INTERFACE I_ControlScheme

END_INTERFACE

(* stored: Version 1.1.0.1, ProductVersion 3.1.4024.6
   Itf I_ControlScheme: Id {f000d3ae-a91a-4047-91a4-fff41840a090} *)
